// TwinCAT 3 PLC project Energy_HB_TSG
// ProgramVersion: 3.1.4023.0
// libraries:
//   Lynus Energy Basic, * (Lynus AG)
//   Lynus Persistent Data V1, * (Lynus AG)
//   Tc2_Standard, * (Beckhoff Automation GmbH)
//   Tc2_System, * (Beckhoff Automation GmbH)
//   Tc3_Module, * (Beckhoff Automation GmbH)
//   TSG Communicator, * (EfficientIO)
// project tree:
//   / Fast.TcTTO, PlcTask.TcTTO, Slow.TcTTO
//   POUs/ prgEM.TcPOU, prgLynusCom.TcPOU, prgLynusVar.TcPOU, prgPersData.TcPOU
// real-time tasks:
//   TASK PlcTask: cycle T#10ms, priority 8, ADS port 350
//   TASK Slow: cycle T#20ms, priority 10, ADS port 351
//   TASK Fast: cycle T#5ms, priority 6, ADS port 352
// I/O:
//   DEVICE Gerät 3 (CX-BK)
//     Box 1 (CX-BK)
// variable links:
//   Energy_HB_TSG/Energy_HB_TSG Instance <-> Device 3 (CX-BK)/Box 1 (CX-BK)
//     PlcTask Inputs/prgEM.fbEM1.fbKL3403.byStateCH1 <-> Term 2 (KL3403)/Channel 1/Status
//     PlcTask Inputs/prgEM.fbEM1.fbKL3403.byStateCH2 <-> Term 2 (KL3403)/Channel 2/Status
//     PlcTask Inputs/prgEM.fbEM1.fbKL3403.byStateCH3 <-> Term 2 (KL3403)/Channel 3/Status
//     PlcTask Inputs/prgEM.fbEM2.fbKL3403.byStateCH1 <-> Term 3 (KL3403)/Channel 1/Status
//     PlcTask Inputs/prgEM.fbEM2.fbKL3403.byStateCH2 <-> Term 3 (KL3403)/Channel 2/Status
//     PlcTask Inputs/prgEM.fbEM2.fbKL3403.byStateCH3 <-> Term 3 (KL3403)/Channel 3/Status
//     PlcTask Inputs/prgEM.fbEM3.fbKL3403.byStateCH1 <-> Term 4 (KL3403)/Channel 1/Status
//     PlcTask Inputs/prgEM.fbEM3.fbKL3403.byStateCH2 <-> Term 4 (KL3403)/Channel 2/Status
//     PlcTask Inputs/prgEM.fbEM3.fbKL3403.byStateCH3 <-> Term 4 (KL3403)/Channel 3/Status
//     PlcTask Inputs/prgEM.fbEM4.fbKL3403.byStateCH1 <-> Term 5 (KL3403)/Channel 1/Status
//     PlcTask Inputs/prgEM.fbEM4.fbKL3403.byStateCH2 <-> Term 5 (KL3403)/Channel 2/Status
//     PlcTask Inputs/prgEM.fbEM4.fbKL3403.byStateCH3 <-> Term 5 (KL3403)/Channel 3/Status
//     PlcTask Inputs/prgEM.fbEM5.fbKL3403.byStateCH1 <-> Term 6 (KL3403)/Channel 1/Status
//     PlcTask Inputs/prgEM.fbEM5.fbKL3403.byStateCH2 <-> Term 6 (KL3403)/Channel 2/Status
//     PlcTask Inputs/prgEM.fbEM5.fbKL3403.byStateCH3 <-> Term 6 (KL3403)/Channel 3/Status
//     PlcTask Inputs/prgEM.fbEM6.fbKL3403.byStateCH1 <-> Term 7 (KL3403)/Channel 1/Status
//     PlcTask Inputs/prgEM.fbEM6.fbKL3403.byStateCH2 <-> Term 7 (KL3403)/Channel 2/Status
//     PlcTask Inputs/prgEM.fbEM6.fbKL3403.byStateCH3 <-> Term 7 (KL3403)/Channel 3/Status
//     PlcTask Inputs/prgEM.fbEM7.fbKL3403.byStateCH1 <-> Term 8 (KL3403)/Channel 1/Status
//     PlcTask Inputs/prgEM.fbEM7.fbKL3403.byStateCH2 <-> Term 8 (KL3403)/Channel 2/Status
//     PlcTask Inputs/prgEM.fbEM7.fbKL3403.byStateCH3 <-> Term 8 (KL3403)/Channel 3/Status
//     PlcTask Inputs/prgEM.fbEM8.fbKL3403.byStateCH1 <-> Term 9 (KL3403)/Channel 1/Status
//     PlcTask Inputs/prgEM.fbEM8.fbKL3403.byStateCH2 <-> Term 9 (KL3403)/Channel 2/Status
//     PlcTask Inputs/prgEM.fbEM8.fbKL3403.byStateCH3 <-> Term 9 (KL3403)/Channel 3/Status
//     PlcTask Inputs/prgEM.fbEM1.fbKL3403.iDataInCH1 <-> Term 2 (KL3403)/Channel 1/Daten Ein
//     PlcTask Inputs/prgEM.fbEM1.fbKL3403.iDataInCH2 <-> Term 2 (KL3403)/Channel 2/Daten Ein
//     PlcTask Inputs/prgEM.fbEM1.fbKL3403.iDataInCH3 <-> Term 2 (KL3403)/Channel 3/Daten Ein
//     PlcTask Inputs/prgEM.fbEM2.fbKL3403.iDataInCH1 <-> Term 3 (KL3403)/Channel 1/Daten Ein
//     PlcTask Inputs/prgEM.fbEM2.fbKL3403.iDataInCH2 <-> Term 3 (KL3403)/Channel 2/Daten Ein
//     PlcTask Inputs/prgEM.fbEM2.fbKL3403.iDataInCH3 <-> Term 3 (KL3403)/Channel 3/Daten Ein
//     PlcTask Inputs/prgEM.fbEM3.fbKL3403.iDataInCH1 <-> Term 4 (KL3403)/Channel 1/Daten Ein
//     PlcTask Inputs/prgEM.fbEM3.fbKL3403.iDataInCH2 <-> Term 4 (KL3403)/Channel 2/Daten Ein
//     PlcTask Inputs/prgEM.fbEM3.fbKL3403.iDataInCH3 <-> Term 4 (KL3403)/Channel 3/Daten Ein
//     PlcTask Inputs/prgEM.fbEM4.fbKL3403.iDataInCH1 <-> Term 5 (KL3403)/Channel 1/Daten Ein
//     PlcTask Inputs/prgEM.fbEM4.fbKL3403.iDataInCH2 <-> Term 5 (KL3403)/Channel 2/Daten Ein
//     PlcTask Inputs/prgEM.fbEM4.fbKL3403.iDataInCH3 <-> Term 5 (KL3403)/Channel 3/Daten Ein
//     PlcTask Inputs/prgEM.fbEM5.fbKL3403.iDataInCH1 <-> Term 6 (KL3403)/Channel 1/Daten Ein
//     PlcTask Inputs/prgEM.fbEM5.fbKL3403.iDataInCH2 <-> Term 6 (KL3403)/Channel 2/Daten Ein
//     PlcTask Inputs/prgEM.fbEM5.fbKL3403.iDataInCH3 <-> Term 6 (KL3403)/Channel 3/Daten Ein
//     PlcTask Inputs/prgEM.fbEM6.fbKL3403.iDataInCH1 <-> Term 7 (KL3403)/Channel 1/Daten Ein
//     PlcTask Inputs/prgEM.fbEM6.fbKL3403.iDataInCH2 <-> Term 7 (KL3403)/Channel 2/Daten Ein
//     PlcTask Inputs/prgEM.fbEM6.fbKL3403.iDataInCH3 <-> Term 7 (KL3403)/Channel 3/Daten Ein
//     PlcTask Inputs/prgEM.fbEM7.fbKL3403.iDataInCH1 <-> Term 8 (KL3403)/Channel 1/Daten Ein
//     PlcTask Inputs/prgEM.fbEM7.fbKL3403.iDataInCH2 <-> Term 8 (KL3403)/Channel 2/Daten Ein
//     PlcTask Inputs/prgEM.fbEM7.fbKL3403.iDataInCH3 <-> Term 8 (KL3403)/Channel 3/Daten Ein
//     PlcTask Inputs/prgEM.fbEM8.fbKL3403.iDataInCH1 <-> Term 9 (KL3403)/Channel 1/Daten Ein
//     PlcTask Inputs/prgEM.fbEM8.fbKL3403.iDataInCH2 <-> Term 9 (KL3403)/Channel 2/Daten Ein
//     PlcTask Inputs/prgEM.fbEM8.fbKL3403.iDataInCH3 <-> Term 9 (KL3403)/Channel 3/Daten Ein
//     PlcTask Inputs/prgEM.fbKBusState.uiKBusState_OUT <-> Inputs/State
//     PlcTask Outputs/prgEM.fbEM1.fbKL3403.byCntrCH1 <-> Term 2 (KL3403)/Channel 1/Kontrolle
//     PlcTask Outputs/prgEM.fbEM1.fbKL3403.byCntrCH2 <-> Term 2 (KL3403)/Channel 2/Kontrolle
//     PlcTask Outputs/prgEM.fbEM1.fbKL3403.byCntrCH3 <-> Term 2 (KL3403)/Channel 3/Kontrolle
//     PlcTask Outputs/prgEM.fbEM2.fbKL3403.byCntrCH1 <-> Term 3 (KL3403)/Channel 1/Kontrolle
//     PlcTask Outputs/prgEM.fbEM2.fbKL3403.byCntrCH2 <-> Term 3 (KL3403)/Channel 2/Kontrolle
//     PlcTask Outputs/prgEM.fbEM2.fbKL3403.byCntrCH3 <-> Term 3 (KL3403)/Channel 3/Kontrolle
//     PlcTask Outputs/prgEM.fbEM3.fbKL3403.byCntrCH1 <-> Term 4 (KL3403)/Channel 1/Kontrolle
//     PlcTask Outputs/prgEM.fbEM3.fbKL3403.byCntrCH2 <-> Term 4 (KL3403)/Channel 2/Kontrolle
//     PlcTask Outputs/prgEM.fbEM3.fbKL3403.byCntrCH3 <-> Term 4 (KL3403)/Channel 3/Kontrolle
//     PlcTask Outputs/prgEM.fbEM4.fbKL3403.byCntrCH1 <-> Term 5 (KL3403)/Channel 1/Kontrolle
//     PlcTask Outputs/prgEM.fbEM4.fbKL3403.byCntrCH2 <-> Term 5 (KL3403)/Channel 2/Kontrolle
//     PlcTask Outputs/prgEM.fbEM4.fbKL3403.byCntrCH3 <-> Term 5 (KL3403)/Channel 3/Kontrolle
//     PlcTask Outputs/prgEM.fbEM5.fbKL3403.byCntrCH1 <-> Term 6 (KL3403)/Channel 1/Kontrolle
//     PlcTask Outputs/prgEM.fbEM5.fbKL3403.byCntrCH2 <-> Term 6 (KL3403)/Channel 2/Kontrolle
//     PlcTask Outputs/prgEM.fbEM5.fbKL3403.byCntrCH3 <-> Term 6 (KL3403)/Channel 3/Kontrolle
//     PlcTask Outputs/prgEM.fbEM6.fbKL3403.byCntrCH1 <-> Term 7 (KL3403)/Channel 1/Kontrolle
//     PlcTask Outputs/prgEM.fbEM6.fbKL3403.byCntrCH2 <-> Term 7 (KL3403)/Channel 2/Kontrolle
//     PlcTask Outputs/prgEM.fbEM6.fbKL3403.byCntrCH3 <-> Term 7 (KL3403)/Channel 3/Kontrolle
//     PlcTask Outputs/prgEM.fbEM7.fbKL3403.byCntrCH1 <-> Term 8 (KL3403)/Channel 1/Kontrolle
//     PlcTask Outputs/prgEM.fbEM7.fbKL3403.byCntrCH2 <-> Term 8 (KL3403)/Channel 2/Kontrolle
//     PlcTask Outputs/prgEM.fbEM7.fbKL3403.byCntrCH3 <-> Term 8 (KL3403)/Channel 3/Kontrolle
//     PlcTask Outputs/prgEM.fbEM8.fbKL3403.byCntrCH1 <-> Term 9 (KL3403)/Channel 1/Kontrolle
//     PlcTask Outputs/prgEM.fbEM8.fbKL3403.byCntrCH2 <-> Term 9 (KL3403)/Channel 2/Kontrolle
//     PlcTask Outputs/prgEM.fbEM8.fbKL3403.byCntrCH3 <-> Term 9 (KL3403)/Channel 3/Kontrolle

CONFIGURATION Energy_HB_TSG
    RESOURCE PLC ON TwinCAT3
        TASK Fast(INTERVAL := T#5ms, PRIORITY := 6);
        TASK PlcTask(INTERVAL := T#10ms, PRIORITY := 8);
        TASK Slow(INTERVAL := T#20ms, PRIORITY := 10);
        PROGRAM prgLynusVar WITH Fast : prgLynusVar;
        PROGRAM prgPersData WITH PlcTask : prgPersData;
        PROGRAM prgEM WITH PlcTask : prgEM;
        PROGRAM prgLynusCom WITH Slow : prgLynusCom;
    END_RESOURCE
END_CONFIGURATION

// ---- POUs/prgLynusVar.TcPOU
PROGRAM prgLynusVar
VAR
	fbVarInfo			: FB_VarInfo;
	fbRW1				: FB_ReadWrite;
	fbRW2				: FB_ReadWrite;
	fbRW3				: FB_ReadWrite;
	fbRW4				: FB_ReadWrite;
	fbRW5				: FB_ReadWrite;
	fbRW6				: FB_ReadWrite;
	fbRW7				: FB_ReadWrite;
	fbRW8				: FB_ReadWrite;
	fbRW9				: FB_ReadWrite;
	fbRW10				: FB_ReadWrite;
	
	FPError				: ARRAY[1..10] OF R_TRIG;
	arrError			: ARRAY[1..10] OF UINT;
END_VAR

fbVarInfo(
	bReadInfo:= , 
	eTMCFile:= eSelectTMCFile.eUseTMCFile, 
	eSavePositionTMCFile:= eSavePositionOnPLC.ePostionC, 
	udiCounterFoundVariables=> , 
	bError=> , 
	bBusy=> , 
	byProgress=> , 
	udiErrorCodeOut=> , 
	eErrorVarInfo_Out=> , 
	sVarWithError=> );
	
fbRW1();
fbRW2();
fbRW3();
fbRW4();
fbRW5();
fbRW6();
fbRW7();
fbRW8();
fbRW9();
fbRW10();


FPError[1](CLK:= fbRW1.bError, Q=> );
FPError[2](CLK:= fbRW2.bError, Q=> );
FPError[3](CLK:= fbRW3.bError, Q=> );
FPError[4](CLK:= fbRW4.bError, Q=> );
FPError[5](CLK:= fbRW5.bError, Q=> );
FPError[6](CLK:= fbRW6.bError, Q=> );
FPError[7](CLK:= fbRW7.bError, Q=> );
FPError[8](CLK:= fbRW8.bError, Q=> );
FPError[9](CLK:= fbRW9.bError, Q=> );
FPError[10](CLK:= fbRW10.bError, Q=> );

IF FPError[1].Q THEN arrError[1] := arrError[1] + 1; END_IF 
IF FPError[2].Q THEN arrError[2] := arrError[2] + 1; END_IF 
IF FPError[3].Q THEN arrError[3] := arrError[3] + 1; END_IF 
IF FPError[4].Q THEN arrError[4] := arrError[4] + 1; END_IF 
IF FPError[5].Q THEN arrError[5] := arrError[5] + 1; END_IF 
IF FPError[6].Q THEN arrError[6] := arrError[6] + 1; END_IF 
IF FPError[7].Q THEN arrError[7] := arrError[7] + 1; END_IF 
IF FPError[8].Q THEN arrError[8] := arrError[8] + 1; END_IF 
IF FPError[9].Q THEN arrError[9] := arrError[9] + 1; END_IF 
IF FPError[10].Q THEN arrError[10] := arrError[10] + 1; END_IF

END_PROGRAM

// ---- POUs/prgPersData.TcPOU
PROGRAM prgPersData
VAR
	fbPersData			: FB_WritePersistentData_CX51x0; 
END_VAR

fbPersData(
	eSaveModeData:= eUSVSaveMode.eSaveWhenPowerfail, 
	bLoadPersistentDataOk=> , 
	bPowerFailDetect=> , 
	bError=> , 
	bySaveProcess=> , 
	dwStorageLast24h=> , 
	udiErrorCode=> );

END_PROGRAM

// ---- POUs/prgEM.TcPOU
PROGRAM prgEM
VAR
	fbKBusState		: FB_K_Bus_State;
	fbEM1			: FB_EM_Beckhoff_KL3403;
	fbEM2			: FB_EM_Beckhoff_KL3403;
	fbEM3			: FB_EM_Beckhoff_KL3403;
	fbEM4			: FB_EM_Beckhoff_KL3403;
	fbEM5			: FB_EM_Beckhoff_KL3403;
	
	wDataL1, wDataL2, wDataL3   AT%I* : WORD;
	bySBL1, bySBL2, bySBL3      AT%I* : BYTE;
	byCBL1, byCBL2, byCBL3      AT%Q*       : BYTE;
	iDataOutL1, iDataOutL2, iDataOutL3  AT%Q* : INT;
	
	fbEM6			: FB_EM_Beckhoff_KL3403;
	fbEM7			: FB_EM_Beckhoff_KL3403;
	fbEM8			: FB_EM_Beckhoff_KL3403;
	fbGrid			: FB_Grid_Power_Ext_Input;			//{#lynus.ag#()}
	lrPowerEM1		: LREAL;							//{#lynus.ag#()}
	lrPowerEM2		: LREAL;							//{#lynus.ag#()}
	lrPowerEM3		: LREAL;							//{#lynus.ag#()}
	lrPowerEM4		: LREAL;							//{#lynus.ag#()}
	lrPowerEM5		: LREAL;							//{#lynus.ag#()}
	lrPowerEM5_1	: LREAL;							//{#lynus.ag#()}
	lrPowerEM5_2	: LREAL;							//{#lynus.ag#()}
	lrPowerEM5_3	: LREAL;							//{#lynus.ag#()}
	lrPowerEM6		: LREAL;							//{#lynus.ag#()}
	lrPowerEM6_1	: LREAL;							//{#lynus.ag#()}
	lrPowerEM6_2	: LREAL;							//{#lynus.ag#()}
	lrPowerEM6_3	: LREAL;							//{#lynus.ag#()}
	lrPowerEM7		: LREAL;							//{#lynus.ag#()}
	lrPowerEM7_1	: LREAL;							//{#lynus.ag#()}
	lrPowerEM7_2	: LREAL;							//{#lynus.ag#()}
	lrPowerEM7_3	: LREAL;							//{#lynus.ag#()}
	lrPowerEM8		: LREAL;							//{#lynus.ag#()}
	lrPowerEM8_1	: LREAL;							//{#lynus.ag#()}
	lrPowerEM8_2	: LREAL;							//{#lynus.ag#()}
	lrPowerEM8_3	: LREAL;							//{#lynus.ag#()}
	lrCounterEM5	: LREAL;							//{#lynus.ag#()}
	lrCounterEM6	: LREAL;							//{#lynus.ag#()}
	lrCounterEM7	: LREAL;							//{#lynus.ag#()}
	lrCounterEM8	: LREAL;							//{#lynus.ag#()}
	
	lrCurrent_EM5_1 : LREAL;							//{#lynus.ag#()}
	lrCurrent_EM5_2 : LREAL;							//{#lynus.ag#()}
	lrCurrent_EM5_3 : LREAL;							//{#lynus.ag#()}
	lrCurrent_EM6_1 : LREAL;							//{#lynus.ag#()}
	lrCurrent_EM6_2 : LREAL;							//{#lynus.ag#()}
	lrCurrent_EM6_3 : LREAL;							//{#lynus.ag#()}
	lrCurrent_EM7_1 : LREAL;							//{#lynus.ag#()}
	lrCurrent_EM7_2 : LREAL;							//{#lynus.ag#()}
	lrCurrent_EM7_3 : LREAL;							//{#lynus.ag#()}
	lrCurrent_EM8_1 : LREAL;							//{#lynus.ag#()}
	lrCurrent_EM8_2 : LREAL;							//{#lynus.ag#()}
	lrCurrent_EM8_3 : LREAL;							//{#lynus.ag#()}
END_VAR

fbKBusState(uiKBusState_OUT=> );


//UV1	
fbEM1(
	bEnable:= TRUE, 
	bChannel1Invers:= TRUE,
	bChannel2Invers:= TRUE,
	bChannel3Invers:= TRUE,
	uiCurrentTransformerRatioL1:= 400, 
	uiCurrentTransformerRatioL2:= 400, 
	uiCurrentTransformerRatioL3:= 400, 
	uiKBusState_IN:= fbKBusState.uiKBusState_OUT, 
	stDataEMPower=> , 
	stDataEMCounter=> , 
	stDataEMPowerRealTime=> , 
	stDataEMCounterRealTime=> , 
	diNrOfEM_OUT=> );

lrPowerEM1 := fbEM1.stDataEMPower.lrPowerTotal;

//UV2	
fbEM2(
	bEnable:= TRUE, 
	bChannel1Invers:= TRUE,
	bChannel2Invers:= TRUE,
	bChannel3Invers:= TRUE,
	uiCurrentTransformerRatioL1:= 400, 
	uiCurrentTransformerRatioL2:= 400, 
	uiCurrentTransformerRatioL3:= 400, 
	uiKBusState_IN:= fbKBusState.uiKBusState_OUT, 
	stDataEMPower=> , 
	stDataEMCounter=> , 
	stDataEMPowerRealTime=> , 
	stDataEMCounterRealTime=> , 
	diNrOfEM_OUT=> );

lrPowerEM2 := fbEM2.stDataEMPower.lrPowerTotal;

//UV3	
fbEM3(
	bEnable:= TRUE, 
	bChannel1Invers:= TRUE,
	bChannel2Invers:= TRUE,
	bChannel3Invers:= TRUE,
	uiCurrentTransformerRatioL1:= 400, 
	uiCurrentTransformerRatioL2:= 400, 
	uiCurrentTransformerRatioL3:= 400, 
	uiKBusState_IN:= fbKBusState.uiKBusState_OUT, 
	stDataEMPower=> , 
	stDataEMCounter=> , 
	stDataEMPowerRealTime=> , 
	stDataEMCounterRealTime=> , 
	diNrOfEM_OUT=> );

lrPowerEM3 := fbEM3.stDataEMPower.lrPowerTotal;	
	
//UV4	
fbEM4(
	bEnable:= TRUE, 
	bChannel1Invers:= TRUE,
	bChannel2Invers:= TRUE,
	bChannel3Invers:= TRUE,
	uiCurrentTransformerRatioL1:= 400, 
	uiCurrentTransformerRatioL2:= 400, 
	uiCurrentTransformerRatioL3:= 400, 
	uiKBusState_IN:= fbKBusState.uiKBusState_OUT, 
	stDataEMPower=> , 
	stDataEMCounter=> , 
	stDataEMPowerRealTime=> , 
	stDataEMCounterRealTime=> , 
	diNrOfEM_OUT=> );

lrPowerEM4 := fbEM4.stDataEMPower.lrPowerTotal;	

//UV5	
fbEM5(
	bEnable:= TRUE, 
	bChannel1Invers:= TRUE,
	bChannel2Invers:= TRUE,
	bChannel3Invers:= TRUE,
	uiCurrentTransformerRatioL1:= 400, 
	uiCurrentTransformerRatioL2:= 400, 
	uiCurrentTransformerRatioL3:= 400, 
	uiKBusState_IN:= fbKBusState.uiKBusState_OUT, 
	stDataEMPower=> , 
	stDataEMCounter=> , 
	stDataEMPowerRealTime=> , 
	stDataEMCounterRealTime=> , 
	diNrOfEM_OUT=> );

lrPowerEM5 := fbEM5.stDataEMPower.lrPowerTotal;	
	lrCounterEM5 := fbEM5.stDataEMCounter.lrTotalCounterEnergy_Consumption;	
		lrPowerEM5_1 := fbEM5.stDataEMPower.lrPowerL1;
			lrPowerEM5_2 := fbEM5.stDataEMPower.lrPowerL2;
				lrPowerEM5_3 := fbEM5.stDataEMPower.lrPowerL3;
					lrCurrent_EM5_1 := fbEM5.stDataEMPower.lrCurrentL1;
						lrCurrent_EM5_2 := fbEM5.stDataEMPower.lrCurrentL2;
							lrCurrent_EM5_3 := fbEM5.stDataEMPower.lrCurrentL3;
	
//UV6
fbEM6(
	bEnable:= TRUE, 
	bChannel1Invers:= TRUE,
	bChannel2Invers:= TRUE,
	bChannel3Invers:= TRUE,
	uiCurrentTransformerRatioL1:= 400, 
	uiCurrentTransformerRatioL2:= 400, 
	uiCurrentTransformerRatioL3:= 400, 
	uiKBusState_IN:= fbKBusState.uiKBusState_OUT, 
	stDataEMPower=> , 
	stDataEMCounter=> , 
	stDataEMPowerRealTime=> , 
	stDataEMCounterRealTime=> , 
	diNrOfEM_OUT=> );

lrPowerEM6 := fbEM6.stDataEMPower.lrPowerTotal;	
	lrCounterEM6 := fbEM6.stDataEMCounter.lrTotalCounterEnergy_Consumption;	
		lrPowerEM6_1 := fbEM6.stDataEMPower.lrPowerL1;
			lrPowerEM6_2 := fbEM6.stDataEMPower.lrPowerL2;
				lrPowerEM6_3 := fbEM6.stDataEMPower.lrPowerL3;
					lrCurrent_EM6_1 := fbEM6.stDataEMPower.lrCurrentL1;
						lrCurrent_EM6_2 := fbEM6.stDataEMPower.lrCurrentL2;
							lrCurrent_EM6_3 := fbEM6.stDataEMPower.lrCurrentL3;
	
//UV7	
fbEM7(
	bEnable:= TRUE, 
	bChannel1Invers:= TRUE,
	bChannel2Invers:= TRUE,
	bChannel3Invers:= TRUE,
	uiCurrentTransformerRatioL1:= 400, 
	uiCurrentTransformerRatioL2:= 400, 
	uiCurrentTransformerRatioL3:= 400, 
	uiKBusState_IN:= fbKBusState.uiKBusState_OUT, 
	stDataEMPower=> , 
	stDataEMCounter=> , 
	stDataEMPowerRealTime=> , 
	stDataEMCounterRealTime=> , 
	diNrOfEM_OUT=> );

lrPowerEM7 := fbEM7.stDataEMPower.lrPowerTotal;
	lrCounterEM7 := fbEM7.stDataEMCounter.lrTotalCounterEnergy_Consumption;	
		lrPowerEM7_1 := fbEM7.stDataEMPower.lrPowerL1;
			lrPowerEM7_2 := fbEM7.stDataEMPower.lrPowerL2;
				lrPowerEM7_3 := fbEM7.stDataEMPower.lrPowerL3;
					lrCurrent_EM7_1 := fbEM7.stDataEMPower.lrCurrentL1;
						lrCurrent_EM7_2 := fbEM7.stDataEMPower.lrCurrentL2;
							lrCurrent_EM7_3 := fbEM7.stDataEMPower.lrCurrentL3;
	
//UV8	
fbEM8(
	bEnable:= TRUE, 
	bChannel1Invers:= TRUE,
	bChannel2Invers:= TRUE,
	bChannel3Invers:= TRUE,
	uiCurrentTransformerRatioL1:= 400, 
	uiCurrentTransformerRatioL2:= 400, 
	uiCurrentTransformerRatioL3:= 400, 
	uiKBusState_IN:= fbKBusState.uiKBusState_OUT, 
	stDataEMPower=> , 
	stDataEMCounter=> , 
	stDataEMPowerRealTime=> , 
	stDataEMCounterRealTime=> , 
	diNrOfEM_OUT=> );

lrPowerEM8 := fbEM8.stDataEMPower.lrPowerTotal;	
	lrCounterEM8 := fbEM8.stDataEMCounter.lrTotalCounterEnergy_Consumption;	
		lrPowerEM8_1 := fbEM8.stDataEMPower.lrPowerL1;
			lrPowerEM8_2 := fbEM8.stDataEMPower.lrPowerL2;
				lrPowerEM8_3 := fbEM8.stDataEMPower.lrPowerL3;
					lrCurrent_EM8_1 := fbEM8.stDataEMPower.lrCurrentL1;
						lrCurrent_EM8_2 := fbEM8.stDataEMPower.lrCurrentL2;
							lrCurrent_EM8_3 := fbEM8.stDataEMPower.lrCurrentL3;
	
//Sum of all 8 Messurements is the Grid power

//Error
IF fbEM5.stDataEMPowerRealTime.byErrorWarning = 2 OR
	fbEM6.stDataEMPowerRealTime.byErrorWarning = 2 OR fbEM7.stDataEMPowerRealTime.byErrorWarning = 2 OR fbEM8.stDataEMPowerRealTime.byErrorWarning = 2 THEN
		fbGrid.bExtErrorGrid := TRUE;
ELSE
		fbGrid.bExtErrorGrid := FALSE;
END_IF	

//Power and Counter Data
fbGrid.lrExtGridPower := fbEM5.stDataEMPowerRealTime.lrPowerTotal +
							fbEM6.stDataEMPowerRealTime.lrPowerTotal + fbEM7.stDataEMPowerRealTime.lrPowerTotal + fbEM8.stDataEMPowerRealTime.lrPowerTotal;

fbGrid.lrExtCounterEnergyT1_Consumption := fbEM5.stDataEMCounterRealTime.lrCounterEnergyT1_Consumption + fbEM6.stDataEMCounterRealTime.lrCounterEnergyT1_Consumption +
													fbEM7.stDataEMCounterRealTime.lrCounterEnergyT1_Consumption + fbEM8.stDataEMCounterRealTime.lrCounterEnergyT1_Consumption;	

fbGrid.lrExtCounterEnergyT2_Consumption := fbEM5.stDataEMCounterRealTime.lrCounterEnergyT2_Consumption + fbEM6.stDataEMCounterRealTime.lrCounterEnergyT2_Consumption +
													fbEM7.stDataEMCounterRealTime.lrCounterEnergyT2_Consumption + fbEM8.stDataEMCounterRealTime.lrCounterEnergyT2_Consumption;							
							
fbGrid.lrExtTotalCounterEnergy_Consumption := fbEM5.stDataEMCounterRealTime.lrTotalCounterEnergy_Consumption + fbEM6.stDataEMCounterRealTime.lrTotalCounterEnergy_Consumption +
													fbEM7.stDataEMCounterRealTime.lrTotalCounterEnergy_Consumption + fbEM8.stDataEMCounterRealTime.lrTotalCounterEnergy_Consumption;
													
fbGrid.lrExtCounterEnergyT1_Production := fbEM5.stDataEMCounterRealTime.lrCounterEnergyT1_Production + fbEM6.stDataEMCounterRealTime.lrCounterEnergyT1_Production +
													fbEM7.stDataEMCounterRealTime.lrCounterEnergyT1_Production + fbEM8.stDataEMCounterRealTime.lrCounterEnergyT1_Production; 
													
fbGrid.lrExtCounterEnergyT2_Production := fbEM5.stDataEMCounterRealTime.lrCounterEnergyT2_Production + fbEM6.stDataEMCounterRealTime.lrCounterEnergyT2_Production +
													fbEM7.stDataEMCounterRealTime.lrCounterEnergyT2_Production + fbEM8.stDataEMCounterRealTime.lrCounterEnergyT2_Production; 
													
fbGrid.lrExtTotalCounterEnergy_Production := fbEM5.stDataEMCounterRealTime.lrTotalCounterEnergy_Production + fbEM6.stDataEMCounterRealTime.lrTotalCounterEnergy_Production +
													fbEM7.stDataEMCounterRealTime.lrTotalCounterEnergy_Production + fbEM8.stDataEMCounterRealTime.lrTotalCounterEnergy_Production;

fbGrid(
	bEnable:= TRUE, 
	diNrOfEMS_IN:= 1, 
	rSizeGridConn:= , 
	bExtErrorGrid:= , 
	lrExtGridPower:= , 
	lrExtTotalCounterEnergy_Consumption:= , 
	lrExtTotalCounterEnergy_Production:= , 
	lrExtCounterEnergyT1_Consumption:= , 
	lrExtCounterEnergyT2_Consumption:= , 
	lrExtCounterEnergyT1_Production:= , 
	lrExtCounterEnergyT2_Production:= , 
	stDataGrid=> , 
	diNrOfGrid_OUT=> );

END_PROGRAM

// ---- POUs/prgLynusCom.TcPOU
PROGRAM prgLynusCom
VAR
	fbCom			: FB_MqttCommunicator;
END_VAR

fbCom(
	bConnect:= TRUE, 
	sUserName:= 'dfe33df1-2501-4272-bd20-2a3c4ced1b25', 
	sUserPassword:= '551afed8-2412-4c45-bca2-67e0714027a0', 
	eSavePositionCertificate:= eSavePositionOnPLC.ePostionC, 
	bConnected=> , 
	bError=> , 
	hrErrorCode=> , 
	eConnectionState=> , 
	eErrorMessage_Out=> );

END_PROGRAM
